// TIA Portal V20 export
TYPE "LER_typeCommunicationSpecialFunctionsStack"
// stored: Access Published
   STRUCT
      specialFunction1 : Bool;
      specialFunction2 : Bool;
      specialFunction3 : Bool;
      specialFunction4 : Bool;
      specialFunction5 : Bool;
      specialFunction6 : Bool;
      specialFunction7 : Bool;
      specialFunction8 : Bool;
      specialFunction9 : Bool;
      specialFunction10 : Bool;
      specialFunction11 : Bool;
      specialFunction12 : Bool;
      specialFunction13 : Bool;
      specialFunction14 : Bool;
      specialFunction15 : Bool;
      specialFunction16 : Bool;
   END_STRUCT;
END_TYPE
